(* CODESYS project Raspi_concat_test.project

Project tree, tasks and I/O mapping:
  Device : CODESYS Control for Raspberry Pi SL, 3S - Smart Software Solutions GmbH, version 3.5.10.20
    application Application
      libraries: Standard, * (System); BASIC, 3.3.3.0 (OSCAT)
      task MainTask (cyclic, interval 4 ms, priority 1) calls PLC_PRG
      program PLC_PRG [ST]
      function block FUOcenControlsCommand [ST]
      data type STlocation
      data type ECommand
    SoftMotion General Axis Pool
    I²C
    SPI
    GPIOs_A_B : GPIOs B+/Pi2, 3S - Smart Software Solutions GmbH, version 1.1.1.10
        unmapped channels: digital inputs (GPIO0..GPIO31), digital outputs (GPIO0..GPIO31)
    Onewire
    Camera device
      <Empty>
*)

// Device/Application/STlocation
TYPE STlocation :
STRUCT
	stlocx : REAL;
	stlocy : REAL;
	sttoolid : INT;
	
END_STRUCT
END_TYPE

// Device/Application/ECommand
TYPE ECommand : (E_AMOV := 1, E_RMOV := 2, E_REL1 := 10, E_REL2 := 20);
END_TYPE

// Device/Application/PLC_PRG
PROGRAM PLC_PRG
VAR
	Locationarray : ARRAY[1..maxbins] OF STlocation;
	Relay01 : FUOcenControlsCommand;
	axistmp : INT := 0;
	
END_VAR
VAR CONSTANT
	maxbins : INT := 60;
END_VAR

Relay01(fuaxis := 1, fucommand := E_AMOV, fup1 := 1, fup2 := 2, fup3 := 3, fuaxisnum := axistmp);

END_PROGRAM

// Device/Application/FUOcenControlsCommand
FUNCTION_BLOCK FUOcenControlsCommand
VAR_INPUT
	fuaxis : INT; (*initial axis*)
	fucommand : Ecommand; (*command type*)
	fuaxisnum : INT := 0; (*amount of axis to process max is 4*)
	fup1 : INT := 0;
	fup2 : INT := 0;
	fup3 : INT := 0;
	fup4 : INT := 0;
	fup5 : INT := 0;
	fup6 : INT := 0;
	fup7 : INT := 0;
END_VAR
VAR_OUTPUT
	fuconstruct : STRING;
	erroron : BOOL := FALSE;
END_VAR
VAR
	i : INT;
	
	futemp : ARRAY[0..maxarray] OF STRING;
	fuempty : STRING;
	imax : INT;
END_VAR
VAR CONSTANT
	fuinitial : STRING := '@'; (*initial char before the axis*)
	fuzero : STRING := '0'; (*used for padding *)
	fucr : STRING := '\R'; (*used for eol in structure*)
	maxaxis : INT := 4;
	maxarray : INT := 10;
END_VAR

(*
	@AA CMND[ X][ Y][ Z][ A]<EOL>[<CS>]
	Square brackets (‘[‘ and ‘]’) indicate parts of the command that are optional. Commands
	should not be sent with square bracket characters in them.
	@ is the at symbol. All commands begin with the at symbol.
	AA is the axis address, 1 to 16. One or more space or tab characters must follow the address.
	CMND is the four character command. The command is not case sensitive.
	[ X][ Y][ Z][ A] is a series of up to four parameters. The number of parameters required
	depends on the command. Parameters must be decimal integer values and cannot contain
	thousands separators. One or more space or tab characters must be present between the
	command and the first parameter, and between each parameter.
	<EOL> is one or more a line-ending characters. Acceptable line-ending characters are carriage
	return (‘\r’ or 0x0D) or newline (‘\n’ or 0x0A).
	
*)

//setup the first two strings in the array
i := 0;
imax := 0;
fuconstruct := fuempty;
CASE fuaxis OF	
	1..9:	futemp[0] := concat(fuinitial,fuzero);
			futemp[0] := concat(futemp[0], INT_TO_STRING(fuaxis));
			imax := 0;
			
	ELSE
			futemp[0] := fuinitial;
			futemp[0] := concat(futemp[0], INT_TO_STRING(fuaxis));
			imax := 0;
END_CASE
//set the parameters according to the command
CASE fucommand OF
	//AMOV command is absolute
	1:	futemp[1] := 'AMOV';
		CASE fuaxisnum OF
			0..1:	futemp[2] := INT_TO_STRING(fup1);
					imax := imax + 2;
			2:		futemp[2] := INT_TO_STRING(fup1);
					futemp[3] := INT_TO_STRING(fup2);
					imax := imax + 3;
			3:		futemp[2] := INT_TO_STRING(fup1);
					futemp[3] := INT_TO_STRING(fup2);
					futemp[4] := INT_TO_STRING(fup3);
					imax := imax +4;
			4:		futemp[2] := INT_TO_STRING(fup1);
					futemp[3] := INT_TO_STRING(fup2);
					futemp[4] := INT_TO_STRING(fup3);
					futemp[5] := INT_TO_STRING(fup4);
					imax := imax +5;
			ELSE
				erroron := TRUE;
		END_CASE
	2:	futemp[1] := 'RMOV';
		CASE fuaxisnum OF
			0..1:	futemp[2] := INT_TO_STRING(fup1);
					imax := imax + 2;
			2:		futemp[2] := INT_TO_STRING(fup1);
					futemp[3] := INT_TO_STRING(fup2);
					imax := imax + 3;
			3:		futemp[2] := INT_TO_STRING(fup1);
					futemp[3] := INT_TO_STRING(fup2);
					futemp[4] := INT_TO_STRING(fup3);
					imax := imax +4;
			4:		futemp[2] := INT_TO_STRING(fup1);
					futemp[3] := INT_TO_STRING(fup2);
					futemp[4] := INT_TO_STRING(fup3);
					futemp[5] := INT_TO_STRING(fup4);
					imax := imax +5;
			ELSE
				erroron := TRUE;
		END_CASE
	10: futemp[1] := 'REL1';
		futemp[2] := INT_TO_STRING(fup1);
		imax := imax + 2;
		
	20: futemp[1] := 'REL2';
		futemp[2] := INT_TO_STRING(fup1);
		imax := imax + 2;
						
END_CASE
FOR i := 0 TO imax DO
	fuconstruct := concat(fuconstruct,futemp[i]);
	fuconstruct := concat(fuconstruct, ' ');
END_FOR
//add the cr
fuconstruct := concat(fuconstruct, fucr);

(*		
		fuconstruct := concat(fuinitial,fuzero);
		fuconstruct := concat(fuconstruct, futemp[0]);
		fuconstruct := concat(fuconstruct, ' ');
		fuconstruct := concat(fuconstruct, 'REL1');
		fuconstruct := concat(fuconstruct, ' ');
		fuconstruct := concat(fuconstruct, futemp[1]);
		fuconstruct := concat(fuconstruct, '$R');
*)

END_FUNCTION_BLOCK
